// TIA Portal V20 export
DATA_BLOCK "LBP_Internal9"   // DB25005
TITLE = Internal DB for basic program / DB interne pour programme de base
// DB only for internal use in the basic program / DB réservé à l'utilisation interne dans le programme de base
// stored: InstanceOfName LBP_InternalProc9, InstanceOfType FB
"LBP_InternalProc9"
   // VAR
   //    statSymbols { ExternalAccessible := 'False'; ExternalVisible := 'False'; ExternalWritable := 'False'} : Array[0..31] of WString;
   //    statResolvedSymbols { ExternalAccessible := 'False'; ExternalVisible := 'False'; ExternalWritable := 'False'} : Array[0..31] of ResolvedSymbol;
   //    InstResolveSymbols { ExternalAccessible := 'False'; ExternalVisible := 'False'; ExternalWritable := 'False'} : ResolveSymbols;
   //    statDestOffsets { ExternalAccessible := 'False'; ExternalVisible := 'False'; ExternalWritable := 'False'} : Array[0..31] of DInt;
   //    statResolveExecute { ExternalAccessible := 'False'; ExternalVisible := 'False'; ExternalWritable := 'False'} : Bool;
   //    statResolveProcessing { ExternalAccessible := 'False'; ExternalVisible := 'False'; ExternalWritable := 'False'} : Bool;
   //    statResolveError { ExternalAccessible := 'False'; ExternalVisible := 'False'; ExternalWritable := 'False'} : Bool;
   //    statResolveStatus { ExternalAccessible := 'False'; ExternalVisible := 'False'; ExternalWritable := 'False'} : Word;
   //    statReResolveNeeded { ExternalAccessible := 'False'; ExternalVisible := 'False'; ExternalWritable := 'False'} : Array[0..31] of Bool;
   // END_VAR
BEGIN
END_DATA_BLOCK
